FUNCTION_BLOCK AXE_plant
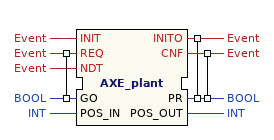
  EVENT_INPUT
    INIT;
    REQ WITH GO;
    NDT;
  END_EVENT
  EVENT_OUTPUT
    INITO WITH PR;
    CNF WITH PR;
  END_EVENT
  VAR_INPUT
    GO : BOOL;
    POS_IN : INT;
  END_VAR
  VAR_OUTPUT
    PR : BOOL;
    POS_OUT : INT;
  END_VAR
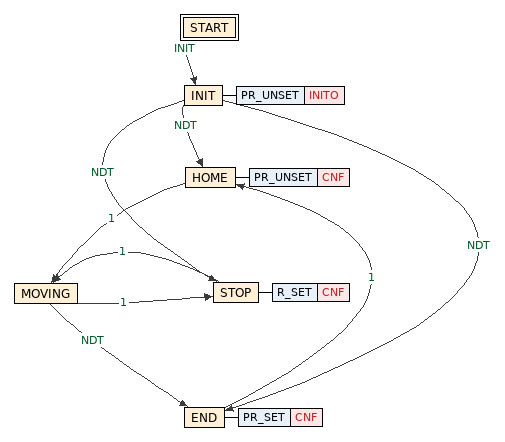
  EC_STATES
    START;
    HOME : PR_UNSET -> CNF;
    MOVING;
    END : PR_SET -> CNF;
    INIT : PR_UNSET -> INITO;
    STOP : R_SET -> CNF;
  END_STATES
  EC_TRANSITIONS
    HOME TO MOVING := 1;
    MOVING TO END := NDT;
    INIT TO HOME := NDT;
    INIT TO END := NDT;
    START TO INIT := INIT;
    END TO HOME := 1;
    MOVING TO STOP := 1;
    STOP TO MOVING := 1;
    INIT TO STOP := NDT;
  END_TRANSITIONS
  ALGORITHM PR_SET IN ST:
PR := TRUE;&#38;#10;POS_OUT := POS_IN;&#38;#10;
  END_ALGORITHM
  ALGORITHM PR_UNSET IN ST:
PR := FALSE;&#38;#10;
  END_ALGORITHM
  ALGORITHM R_SET IN ST:
POS_OUT := 5;&#38;#10;
  END_ALGORITHM
END_FUNCTION_BLOCK
